PROGRAM MAIN
VAR
END_VAR

END_PROGRAM

(* stored: Version 1.1.0.1
   POU MAIN: Id {21f3a158-4837-47ff-8ec7-29454a44967d} *)
